// TIA Portal V15.1 export
// export: Created 2020-06-12T07:35:55.7724609Z, ExportSetting None, DisplayName Totally Integrated Automation Portal, DisplayVersion V15.1, DisplayName TIA Portal Openness, DisplayVersion V15.1, DisplayName STEP 7 Professional, DisplayVersion V15.1, DisplayName STEP 7 Safety, DisplayVersion V15.1, DisplayName WinCC Advanced, DisplayVersion V15.1
FUNCTION "SLAG_dose" : Void   // FC161, FBD
TITLE = Slag addition rated loading (dosing) control
{ S7_Optimized_Access := 'TRUE' }
// stored: SetENOAutomatically False
   VAR_TEMP
      tActualRate : Real;
   END_VAR
BEGIN

REGION Network 1: An actual feeding rate calculation [kg/min]
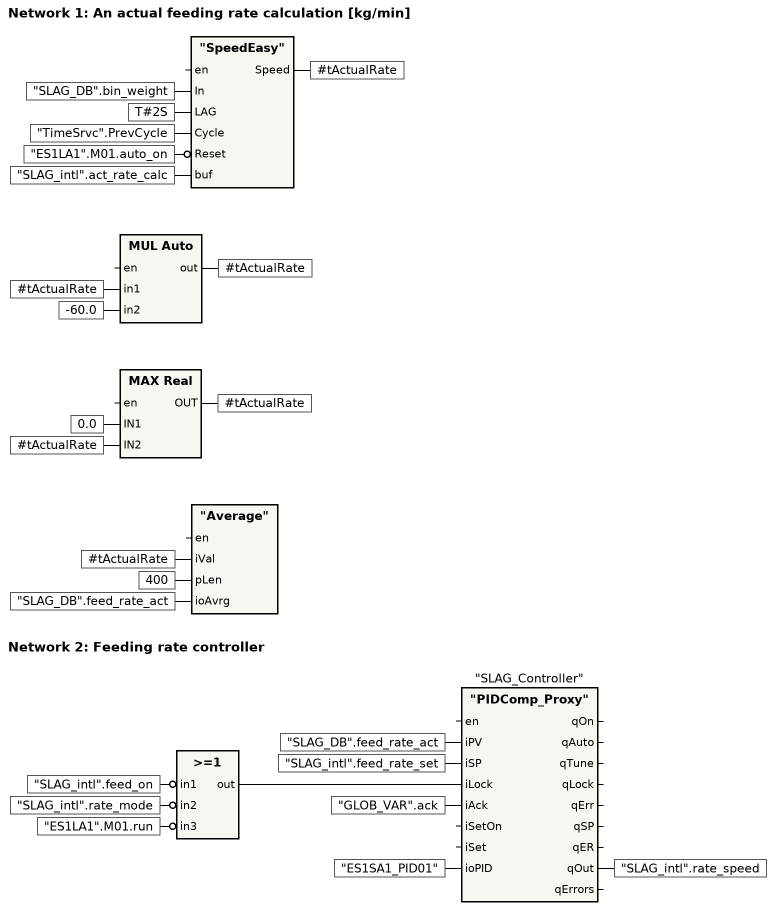
   "SpeedEasy"(In := "SLAG_DB".bin_weight,
               LAG := T#2S,
               Cycle := "TimeSrvc".PrevCycle,
               Reset := NOT "ES1LA1".M01.auto_on,
               buf := "SLAG_intl".act_rate_calc,
               Speed => #tActualRate);
   #tActualRate := #tActualRate * (-60.0);
   #tActualRate := MAX(IN1 := 0.0, IN2 := #tActualRate);
   "Average"(iVal := #tActualRate, pLen := 400, ioAvrg := "SLAG_DB".feed_rate_act);
END_REGION

REGION Network 2: Feeding rate controller
   // #tActualRate =>  "SLAG_DB".feed_rate_act
   "SLAG_Controller"(iPV := "SLAG_DB".feed_rate_act,   // "PIDComp_Proxy"
                     iSP := "SLAG_intl".feed_rate_set,
                     iLock := NOT "SLAG_intl".feed_on OR NOT "SLAG_intl".rate_mode OR NOT "ES1LA1".M01.run,
                     iAck := "GLOB_VAR".ack,
                     ioPID := "ES1SA1_PID01",
                     qOut => "SLAG_intl".rate_speed);
END_REGION
END_FUNCTION
